(*

## Short summary

This class provides assert statements for unsigned integers from 8~64 bit length 
It implements the interface `IUnsignedIntegerAssertions`
For 8 bit intgers use `UnsignedIntegerAssertions.short`
For 16 bit intgers use `UnsignedIntegerAssertions.simple`
For 32 bit intgers use `UnsignedIntegerAssertions.double`
For 64 bit intgers use `UnsignedIntegerAssertions.long`
For integers in register length use `UnsignedIntegerAssertions.x`

.. <legal notes>

legal notes
=================
| SPDX-FileCopyrightText: © 2022 ekvip automation GmbH <info@ekvip.de>
| SPDX-License-Identifier: Apache-2.0
| For details check: Apache-2.0_

.. _Apache-2.0: https://www.apache.org/licenses/LICENSE-2.0

.. </legal notes>



*)

{attribute 'reflection'}
FUNCTION_BLOCK INTERNAL UnsignedIntegerAssertions EXTENDS CNM_AbstractObject.Object IMPLEMENTS IUnsignedIntegerAssertions
VAR
	(* class to handle assert statements for unsigned short integers *)
	usintAssertions	:UsintAssertions();
	(* class to handle assert statements for unsigned integers *)
	uintAssertions	:UintAssertions();
	(* class to handle assert statements for unsigned double integers *)
	udintAssertions	:UdintAssertions();
	(* class to handle assert statements for unsigned register length integers *)
	uxintAssertions	:UxintAssertions();
	(* class to handle assert statements for unsigned long integers *)
	ulintAssertions	:UlintAssertions();
END_VAR

(*

## Short summary
This abstract property returns the class name of the concrete object, 
It's for debugging purpose

.. <legal notes>

legal notes
=================
| SPDX-FileCopyrightText: © 2022 ekvip automation GmbH <info@ekvip.de>
| SPDX-License-Identifier: Apache-2.0
| For details check: Apache-2.0_

.. _Apache-2.0: https://www.apache.org/licenses/LICENSE-2.0

.. </legal notes>

*)

PROPERTY className :CNM_AbstractObject.ClassName
GET
className := 'CNM_Assertor.UnsignedIntegerAssertions';
END_GET
END_PROPERTY

(*

## Short summary
Returns the interface `IUdintAssertions` with assert statements for unsigned 32 bit integers 

.. <legal notes>

legal notes
=================
| SPDX-FileCopyrightText: © 2022 ekvip automation GmbH <info@ekvip.de>
| SPDX-License-Identifier: Apache-2.0
| For details check: Apache-2.0_

.. _Apache-2.0: https://www.apache.org/licenses/LICENSE-2.0

.. </legal notes>

*)

PROPERTY double :IUdintAssertions
GET
double := THIS^.udintAssertions;
END_GET
END_PROPERTY

(*

## Short summary
Returns the interface `IUlintAssertions` with assert statements for unsigned 64 bit integers 

.. <legal notes>

legal notes
=================
| SPDX-FileCopyrightText: © 2022 ekvip automation GmbH <info@ekvip.de>
| SPDX-License-Identifier: Apache-2.0
| For details check: Apache-2.0_

.. _Apache-2.0: https://www.apache.org/licenses/LICENSE-2.0

.. </legal notes>

*)

PROPERTY long :IUlintAssertions
GET
long := THIS^.ulintAssertions;
END_GET
END_PROPERTY

(*

## Short summary
This methods is the setter for the callback class if an assertion was false

.. <legal notes>

legal notes
=================
| SPDX-FileCopyrightText: © 2022 ekvip automation GmbH <info@ekvip.de>
| SPDX-License-Identifier: Apache-2.0
| For details check: Apache-2.0_

.. _Apache-2.0: https://www.apache.org/licenses/LICENSE-2.0

.. </legal notes>



*)

METHOD setCallBack
VAR_INPUT
	(* the class that must be informed if an assertion is false *)
	callBack	:IAssertCallBack;  
END_VAR
THIS^.usintAssertions.setCallBack(callBack);
THIS^.uintAssertions.setCallBack(callBack);
THIS^.udintAssertions.setCallBack(callBack);
THIS^.uxintAssertions.setCallBack(callBack);
THIS^.ulintAssertions.setCallBack(callBack);
END_METHOD

(*

## Short summary
Returns the interface `IUsintAssertions` with assert statements for unsigned 8 bit integers 

.. <legal notes>

legal notes
=================
| SPDX-FileCopyrightText: © 2022 ekvip automation GmbH <info@ekvip.de>
| SPDX-License-Identifier: Apache-2.0
| For details check: Apache-2.0_

.. _Apache-2.0: https://www.apache.org/licenses/LICENSE-2.0

.. </legal notes>

*)

PROPERTY short :IUsintAssertions
GET
short := THIS^.usintAssertions;
END_GET
END_PROPERTY

(*

## Short summary
Returns the interface `IUintAssertions` with assert statements for unsigned 16 bit integers 

.. <legal notes>

legal notes
=================
| SPDX-FileCopyrightText: © 2022 ekvip automation GmbH <info@ekvip.de>
| SPDX-License-Identifier: Apache-2.0
| For details check: Apache-2.0_

.. _Apache-2.0: https://www.apache.org/licenses/LICENSE-2.0

.. </legal notes>

*)

PROPERTY simple :IUintAssertions
GET
simple := THIS^.uintAssertions;
END_GET
END_PROPERTY

(*

## Short summary
Returns the interface `IUxintAssertions` with assert statements for unsigned integers register length 

.. <legal notes>

legal notes
=================
| SPDX-FileCopyrightText: © 2022 ekvip automation GmbH <info@ekvip.de>
| SPDX-License-Identifier: Apache-2.0
| For details check: Apache-2.0_

.. _Apache-2.0: https://www.apache.org/licenses/LICENSE-2.0

.. </legal notes>

*)

PROPERTY x :IUxintAssertions
GET
x := THIS^.uxintAssertions;
END_GET
END_PROPERTY

END_FUNCTION_BLOCK

(* stored: Version 1.1.0.1, ProductVersion 3.1.4026.12
   POU UnsignedIntegerAssertions: Id {d26d2d05-0d86-4837-8178-4e02e7d3d780}, SpecialFunc None
   Property className: Id {e8ab4c70-40a2-4660-bc50-a670906e80ff}
   Get Get: Id {3fa71b51-3f22-4b14-995c-0306e7ed152f}
   Property double: Id {0b4db36d-1d7e-4d25-b3c5-0ccd390d6639}
   Get Get: Id {7c990063-2502-416f-adc8-265bd1037562}
   Property long: Id {7aa11f53-2289-4f5f-ab40-9dc9506ab775}
   Get Get: Id {c68bd8bd-8cf6-497e-8cea-1564dea08408}
   Method setCallBack: Id {145eb7fa-8974-4bd9-b18b-3e0d74cd9984}
   Property short: Id {9160085d-91ac-4c1c-a84f-d3e2ff342b1c}
   Get Get: Id {a0ec1e1d-bf72-4951-8ce2-1a0efd4fbcec}
   Property simple: Id {b73e7c32-727b-4d75-891c-563b36a028d3}
   Get Get: Id {272da927-4366-495c-a1e8-a79d8c288246}
   Property x: Id {baedee3b-e75c-495b-8ed9-6238b278e602}
   Get Get: Id {a0c5b920-c10a-4e6f-a867-dbd8f53eb59e} *)
